FUNCTION AjustarIndice : INT
VAR_INPUT
    ValorBase: INT;
END_VAR					//Cambiar por un Property?

IF ValorBase < 1 THEN
    AjustarIndice := ValorBase + 8;
ELSE
    AjustarIndice := ValorBase;
END_IF

END_FUNCTION

(* stored: Version 1.1.0.1, ProductVersion 3.1.4024.12
   POU AjustarIndice: Id {38e6a205-0c79-4781-b76a-9d4083be1a45}, SpecialFunc None *)
